// This function Block extends the Referenced Library Mover (FB), so the user can expand the capabilities of the XTS Mover Functions
FUNCTION_BLOCK ApplicationMover EXTENDS Mover
VAR_INPUT
END_VAR
VAR_OUTPUT
END_VAR
VAR
	cnt: UDINT;
	_PositionLag: LREAL;
	fbMC_CalcDynamicsByRampTime: MC_CalcDynamicsByRampTime;
END_VAR

METHOD Cyclic : iMover
VAR_IN_OUT
	GroupReference	: AXES_GROUP_REF;
END_VAR
// Call Base Class (Mover) Cyclic Logic
SUPER^.Cyclic(GroupReference);

//======= 
// To Call ApplicationMover addon Method/Properties/Variables... 
//		you must call Mover[] array index directly, as Station/Zone/PositionTrig/SpeedTrig do not know about ApplicationMover add ons

// Add ApplicationMover specific code here
cnt:= cnt + 1;
_PositionLag:= THIS^.AxisReference.NcToPlc.PosDiff;
END_METHOD

METHOD MoveToStationByRampTime
VAR_INPUT
	DestinationStation	: REFERENCE TO Station;	
    Velocity     : LREAL;
    RampTime     : LREAL;
    Stiffness    : LREAL;
	Gap			 : LREAL;
END_VAR
VAR
	MotionParameters: MotionParameters_typ;
END_VAR
// This method internally calls MC_CalcDynamicsByRampTime from Tc2_MC2.lib
// https://infosys.beckhoff.com/content/1033/tcplclib_tc2_mc2/13611300875.html?id=1298283191705576852

fbMC_CalcDynamicsByRampTime(
	Velocity:= Velocity, 
	RampTime:= RampTime, 
	Stiffness:= Stiffness, 
	Error=> , 
	ErrorID=> , 
	Acceleration=> , 
	Deceleration=> , 
	Jerk=> );

MotionParameters.Velocity			:= Velocity;
MotionParameters.Acceleration		:= fbMC_CalcDynamicsByRampTime.Acceleration;
MotionParameters.Deceleration		:= fbMC_CalcDynamicsByRampTime.Deceleration;
MotionParameters.Jerk				:= fbMC_CalcDynamicsByRampTime.Jerk;
MotionParameters.Gap				:= Gap;
MotionParameters.Direction			:= Tc2_Mc2.MC_Direction.MC_Positive_Direction;

SUPER^.MotionParameters:= MotionParameters;
SUPER^.MoveToStation(DestinationStation);
END_METHOD

{attribute 'monitoring' := 'call'}
PROPERTY PositionLag : LREAL
GET
PositionLag:= _PositionLag;
END_GET
END_PROPERTY

END_FUNCTION_BLOCK

(* stored: Version 1.1.0.1, ProductVersion 3.1.4026.8
   POU ApplicationMover: Id {516536b5-5233-0a95-01e8-9585147c75fa}, SpecialFunc None
   Method Cyclic: Id {a81886a0-983c-0294-0adc-9591fa48a449}
   Method MoveToStationByRampTime: Id {30fb390b-b4a8-0444-29f0-600dae10b753}
   Property PositionLag: Id {2f9b4da0-9f46-0501-2862-3b56ba7816bb}
   Get Get: Id {8ea91099-3f22-02ba-0930-a3b600f2f5d6} *)
